TYPE "UDT_ZC_DISP_TONR"
VERSION : 0.1
   STRUCT
      SP : Int := 5;
      ET : Int := 0;
      RT : Int := 0;
      IN : Bool := FALSE;
      Q : Bool := FALSE;
      RESET : Bool := FALSE;
   END_STRUCT;

END_TYPE

